// TIA Portal project "Project1" (V16)

(* hardware
DEVICE "S71500/ET200MP station_1"  S7-1500 station
   slot 0: "Rail_0"  Rack  6ES7 590-1***0-0AA0
   slot 1: "PLC_1"  CPU 1512C-1 PN  6ES7 512-1CK00-0AB0  V2.1
      slot 3: "CPU display_1"  6ES7591-1AA00-0AA0
      slot 32768: "PROFINET interface_1"  X1
         slot 32769: "Port_1"  X1 P1
         slot 32770: "Port_2"  X1 P2
*)

// ===== PLC "PLC_1"  CPU 1512C-1 PN =====

VAR_GLOBAL   // PLC tag table "Default tag table"
   "Blueprint Input 01" AT %I10.0 : Bool;   // Optic Sensor - G1BG1
   "Blueprint Input 02" AT %I10.1 : Bool;   // Optic Sensor - G1BG2
   "Blueprint Input 03" AT %I10.2 : Bool;   // Optic Sensor - G1BG3
   "Blueprint Input 04" AT %I10.3 : Bool;   // Optic Sensor - G1BG4
   "Blueprint Input 05" AT %I10.4 : Bool;   // Optic Sensor - G2BG1
   "Blueprint Input 06" AT %I10.5 : Bool;
   "Blueprint Input 07" AT %I10.6 : Bool;   // Optic Sensor - G2BG3
   "Blueprint Input 08" AT %I10.7 : Bool;
   "Blueprint Output 01" AT %Q4.0 : Bool;   // Treadmill Floor Actuator - G1XG1-X1
   "Blueprint Output 02" AT %Q4.1 : Bool;   // Treadmill Floor Actuator - G1XG1-X1 - Reverse
   "Blueprint Output 03" AT %Q4.2 : Bool;   // Threadmill Arm Actuator - G1MB1
   "Blueprint Output 04" AT %Q4.3 : Bool;   // Threadmill Blocker Piston Actuator - G1MB2
   "Blueprint Output 05" AT %Q4.4 : Bool;   // Threadmill Floor Actuator - G2XG1
   "Blueprint Output 06" AT %Q4.5 : Bool;   // Threadmill Floor Actuator - G2XG1 - Reverse
   "Blueprint Output 07" AT %Q4.6 : Bool;
   "Blueprint Output 08" AT %Q4.7 : Bool;
   "Pannel Input 01" AT %I11.0 : Bool;   // Start Button
   "Pannel Input 02" AT %I11.1 : Bool;   // Stop Button
   "Pannel Input 03" AT %I11.2 : Bool;   // Auto/Man Key
   "Pannel Input 04" AT %I11.3 : Bool;   // Reset Button
   "Pannel Input 05" AT %I11.4 : Bool;
   "Pannel Input 06" AT %I11.5 : Bool;   // "Stop the world"/"Panic"/"Emergency Stop" Button
   "Pannel Input 07" AT %I11.6 : Bool;
   "Pannel Input 08" AT %I11.7 : Bool;
   "Pannel Output 01" AT %Q5.0 : Bool;   // LED - Start Button
   "Pannel Output 02" AT %Q5.1 : Bool;   // LED - Stop Button
   "Pannel Output 03" AT %Q5.2 : Bool;   // LED - Q1
   "Pannel Output 04" AT %Q5.3 : Bool;   // LED - Q2
   "Pannel Output 05" AT %Q5.4 : Bool;
   "Pannel Output 06" AT %Q5.5 : Bool;
   "Pannel Output 07" AT %Q5.6 : Bool;
   "Pannel Output 08" AT %Q5.7 : Bool;
   "Blueprint ON Signal" AT %M5000.0 : Bool;
END_VAR

// folder: System blocks/Program resources

DATA_BLOCK "Blueprint ON Pulse"   // DB1
{ S7_Optimized_Access := 'TRUE' }
AUTHOR : Simatic
FAMILY : IEC
NAME : IEC_TMR
VERSION : 1.0
// stored: InstanceOfName IEC_TIMER
"IEC_TIMER"
BEGIN
END_DATA_BLOCK

// folder: (top level)

ORGANIZATION_BLOCK "Main"   // OB1, LAD, ProgramCycle
TITLE = "Main Program Sweep (Cycle)"
{ S7_Optimized_Access := 'TRUE' }
VERSION : 0.1
   VAR_INPUT
      Initial_Call : Bool;   // Initial call of this OB
      Remanence : Bool;   // =True, if remanent data are available
   END_VAR
BEGIN

REGION Network 1: LED - Q1
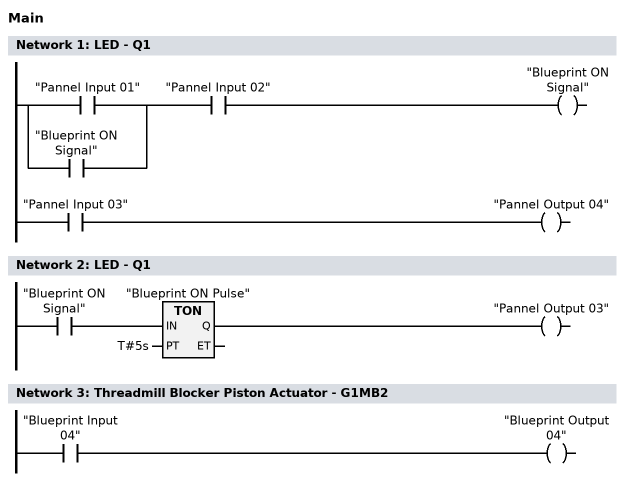
   RUNG wire#powerrail
      Contact( "Pannel Input 01" )
      wire#w1
      Contact( "Pannel Input 02" )
      Coil( "Blueprint ON Signal" )
   END_RUNG
   RUNG wire#powerrail
      Contact( "Blueprint ON Signal" )
   END_RUNG wire#w1
   RUNG wire#powerrail
      Contact( "Pannel Input 03" )
      Coil( "Pannel Output 04" )
   END_RUNG
   // the same network as SCL:
   "Blueprint ON Signal" := ("Pannel Input 01" OR "Blueprint ON Signal") AND "Pannel Input 02";
   "Pannel Output 04" := "Pannel Input 03";
END_REGION

REGION Network 2: LED - Q1
   "Blueprint ON Pulse".TON(IN := "Blueprint ON Signal", PT := T#5s);
   "Pannel Output 03" := "Blueprint ON Pulse".Q;
END_REGION

REGION Network 3: Threadmill Blocker Piston Actuator - G1MB2
   RUNG wire#powerrail
      Contact( "Blueprint Input 04" )
      Coil( "Blueprint Output 04" )
   END_RUNG
   // the same network as SCL:
   "Blueprint Output 04" := "Blueprint Input 04";
END_REGION
END_ORGANIZATION_BLOCK